// TIA Portal V17 export
// export: Created 2025-05-08T13:17:39.9382166Z, ExportSetting WithDefaults, DisplayName Totally Integrated Automation Portal, DisplayVersion V17 Update 8, DisplayName TIA Portal Openness, DisplayVersion V17 Update 8, DisplayName TIA Portal Version Control Interface, DisplayVersion V17, DisplayName SINAMICS Startdrive Advanced, DisplayVersion V17 SP2, DisplayName SINAMICS Startdrive G110M, G120, G120C, G120D, G120P, G115D, DisplayVersion V17 SP2, DisplayName SINAMICS Startdrive G130, G150, S120, S150, SINAMICS MV, S210, DisplayVersion V17 SP2, DisplayName STEP 7 Professional, DisplayVersion V17 Update 8, DisplayName SINUMERIK ONE STEP 7 Toolbox, DisplayVersion V17 Update 12, DisplayName SINUMERIK 840D sl STEP 7 Toolbox, DisplayVersion V17 Update 12, DisplayName STEP 7 Safety, DisplayVersion V17 Update 6, DisplayName WinCC Advanced, DisplayVersion V17 Update 8
FUNCTION "FC2011_STEP_BY_STEP_MODE" : Void   // FC2011, LAD
{ S7_Optimized_Access := 'FALSE' }
AUTHOR : ETXETAR
VERSION : 1.0
// stored: AutoNumber false, IsIECCheckEnabled false, SetENOAutomatically false, UDAEnableTagReadback false
   VAR CONSTANT
      FC_NUMBER : DInt := 2011;
   END_VAR
   VAR_TEMP   // added for the SCL form of the ladder/FBD networks
      _w1 : Bool;
      _w2 : Bool;
   END_VAR
BEGIN

REGION Network 1: GENERAL CONDITIONS
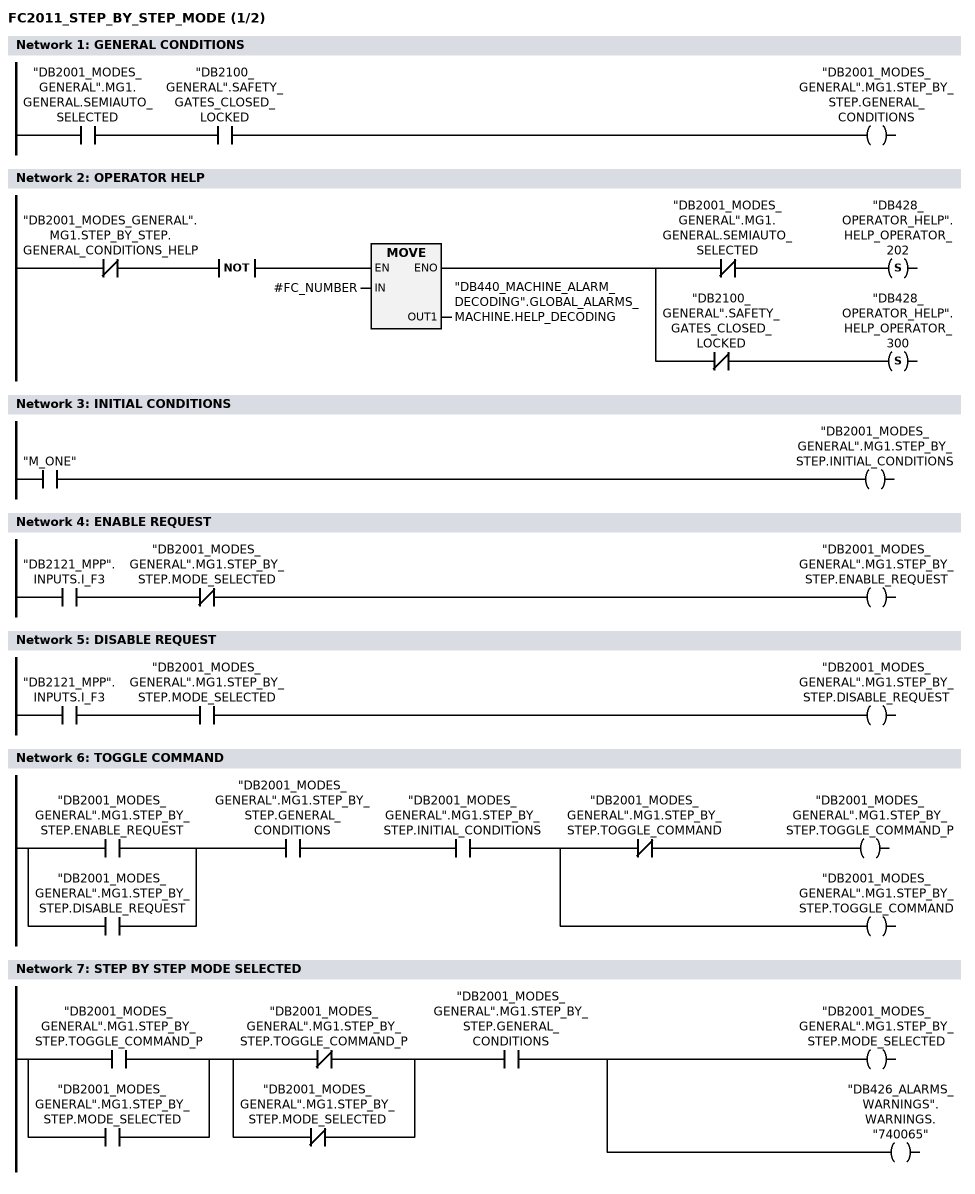
   RUNG wire#powerrail
      Contact( "DB2001_MODES_GENERAL".MG1.GENERAL.SEMIAUTO_SELECTED )
      Contact( "DB2100_GENERAL".SAFETY_GATES_CLOSED_LOCKED )
      Coil( "DB2001_MODES_GENERAL".MG1.STEP_BY_STEP.GENERAL_CONDITIONS )
   END_RUNG
   // the same network as SCL:
   "DB2001_MODES_GENERAL".MG1.STEP_BY_STEP.GENERAL_CONDITIONS := "DB2001_MODES_GENERAL".MG1.GENERAL.SEMIAUTO_SELECTED AND "DB2100_GENERAL".SAFETY_GATES_CLOSED_LOCKED;
END_REGION

REGION Network 2: OPERATOR HELP
   RUNG wire#powerrail
      I_Contact( "DB2001_MODES_GENERAL".MG1.STEP_BY_STEP.GENERAL_CONDITIONS_HELP )
      Not()
      { S7_GenerateENO := "TRUE" } Move(in := #FC_NUMBER, out1 => "DB440_MACHINE_ALARM_DECODING".GLOBAL_ALARMS_MACHINE.HELP_DECODING)
      wire#w1
      I_Contact( "DB2001_MODES_GENERAL".MG1.GENERAL.SEMIAUTO_SELECTED )
      S_Coil( "DB428_OPERATOR_HELP".HELP_OPERATOR_202 )
   END_RUNG
   RUNG wire#w1
      I_Contact( "DB2100_GENERAL".SAFETY_GATES_CLOSED_LOCKED )
      S_Coil( "DB428_OPERATOR_HELP".HELP_OPERATOR_300 )
   END_RUNG
   // the same network as SCL:
   // ENO of a box is taken as its EN; it also drops when the box reports an error
   #_w1 := NOT (NOT "DB2001_MODES_GENERAL".MG1.STEP_BY_STEP.GENERAL_CONDITIONS_HELP);
   IF #_w1 THEN "DB440_MACHINE_ALARM_DECODING".GLOBAL_ALARMS_MACHINE.HELP_DECODING := #FC_NUMBER; END_IF;
   IF #_w1 AND NOT "DB2001_MODES_GENERAL".MG1.GENERAL.SEMIAUTO_SELECTED THEN
       "DB428_OPERATOR_HELP".HELP_OPERATOR_202 := TRUE;
   END_IF;
   IF #_w1 AND NOT "DB2100_GENERAL".SAFETY_GATES_CLOSED_LOCKED THEN
       "DB428_OPERATOR_HELP".HELP_OPERATOR_300 := TRUE;
   END_IF;
END_REGION

REGION Network 3: INITIAL CONDITIONS
   RUNG wire#powerrail
      Contact( "M_ONE" )
      Coil( "DB2001_MODES_GENERAL".MG1.STEP_BY_STEP.INITIAL_CONDITIONS )
   END_RUNG
   // the same network as SCL:
   "DB2001_MODES_GENERAL".MG1.STEP_BY_STEP.INITIAL_CONDITIONS := "M_ONE";
END_REGION

REGION Network 4: ENABLE REQUEST
   RUNG wire#powerrail
      Contact( "DB2121_MPP".INPUTS.I_F3 )
      I_Contact( "DB2001_MODES_GENERAL".MG1.STEP_BY_STEP.MODE_SELECTED )
      Coil( "DB2001_MODES_GENERAL".MG1.STEP_BY_STEP.ENABLE_REQUEST )
   END_RUNG
   // the same network as SCL:
   "DB2001_MODES_GENERAL".MG1.STEP_BY_STEP.ENABLE_REQUEST := "DB2121_MPP".INPUTS.I_F3 AND NOT "DB2001_MODES_GENERAL".MG1.STEP_BY_STEP.MODE_SELECTED;
END_REGION

REGION Network 5: DISABLE REQUEST
   RUNG wire#powerrail
      Contact( "DB2121_MPP".INPUTS.I_F3 )
      Contact( "DB2001_MODES_GENERAL".MG1.STEP_BY_STEP.MODE_SELECTED )
      Coil( "DB2001_MODES_GENERAL".MG1.STEP_BY_STEP.DISABLE_REQUEST )
   END_RUNG
   // the same network as SCL:
   "DB2001_MODES_GENERAL".MG1.STEP_BY_STEP.DISABLE_REQUEST := "DB2121_MPP".INPUTS.I_F3 AND "DB2001_MODES_GENERAL".MG1.STEP_BY_STEP.MODE_SELECTED;
END_REGION

REGION Network 6: TOGGLE COMMAND
   RUNG wire#powerrail
      Contact( "DB2001_MODES_GENERAL".MG1.STEP_BY_STEP.ENABLE_REQUEST )
      wire#w1
      Contact( "DB2001_MODES_GENERAL".MG1.STEP_BY_STEP.GENERAL_CONDITIONS )
      Contact( "DB2001_MODES_GENERAL".MG1.STEP_BY_STEP.INITIAL_CONDITIONS )
      wire#w2
      I_Contact( "DB2001_MODES_GENERAL".MG1.STEP_BY_STEP.TOGGLE_COMMAND )
      Coil( "DB2001_MODES_GENERAL".MG1.STEP_BY_STEP.TOGGLE_COMMAND_P )
   END_RUNG
   RUNG wire#powerrail
      Contact( "DB2001_MODES_GENERAL".MG1.STEP_BY_STEP.DISABLE_REQUEST )
   END_RUNG wire#w1
   RUNG wire#w2
      Coil( "DB2001_MODES_GENERAL".MG1.STEP_BY_STEP.TOGGLE_COMMAND )
   END_RUNG
   // the same network as SCL:
   #_w1 := ("DB2001_MODES_GENERAL".MG1.STEP_BY_STEP.ENABLE_REQUEST OR "DB2001_MODES_GENERAL".MG1.STEP_BY_STEP.DISABLE_REQUEST) AND "DB2001_MODES_GENERAL".MG1.STEP_BY_STEP.GENERAL_CONDITIONS AND "DB2001_MODES_GENERAL".MG1.STEP_BY_STEP.INITIAL_CONDITIONS;
   "DB2001_MODES_GENERAL".MG1.STEP_BY_STEP.TOGGLE_COMMAND_P := #_w1 AND NOT "DB2001_MODES_GENERAL".MG1.STEP_BY_STEP.TOGGLE_COMMAND;
   "DB2001_MODES_GENERAL".MG1.STEP_BY_STEP.TOGGLE_COMMAND := #_w1;
END_REGION

REGION Network 7: STEP BY STEP MODE SELECTED
   RUNG wire#powerrail
      Contact( "DB2001_MODES_GENERAL".MG1.STEP_BY_STEP.TOGGLE_COMMAND_P )
      wire#w1
      I_Contact( "DB2001_MODES_GENERAL".MG1.STEP_BY_STEP.TOGGLE_COMMAND_P )
      wire#w2
      Contact( "DB2001_MODES_GENERAL".MG1.STEP_BY_STEP.GENERAL_CONDITIONS )
      wire#w3
      Coil( "DB2001_MODES_GENERAL".MG1.STEP_BY_STEP.MODE_SELECTED )
   END_RUNG
   RUNG wire#powerrail
      Contact( "DB2001_MODES_GENERAL".MG1.STEP_BY_STEP.MODE_SELECTED )
   END_RUNG wire#w1
   RUNG wire#w1
      I_Contact( "DB2001_MODES_GENERAL".MG1.STEP_BY_STEP.MODE_SELECTED )
   END_RUNG wire#w2
   RUNG wire#w3
      Coil( "DB426_ALARMS_WARNINGS".WARNINGS."740065" )
   END_RUNG
   // the same network as SCL:
   "DB2001_MODES_GENERAL".MG1.STEP_BY_STEP.MODE_SELECTED := ("DB2001_MODES_GENERAL".MG1.STEP_BY_STEP.TOGGLE_COMMAND_P OR "DB2001_MODES_GENERAL".MG1.STEP_BY_STEP.MODE_SELECTED) AND (NOT "DB2001_MODES_GENERAL".MG1.STEP_BY_STEP.TOGGLE_COMMAND_P OR NOT "DB2001_MODES_GENERAL".MG1.STEP_BY_STEP.MODE_SELECTED) AND "DB2001_MODES_GENERAL".MG1.STEP_BY_STEP.GENERAL_CONDITIONS;
   "DB426_ALARMS_WARNINGS".WARNINGS."740065" := "DB2001_MODES_GENERAL".MG1.STEP_BY_STEP.MODE_SELECTED;
END_REGION

REGION Network 8: WARNINGS
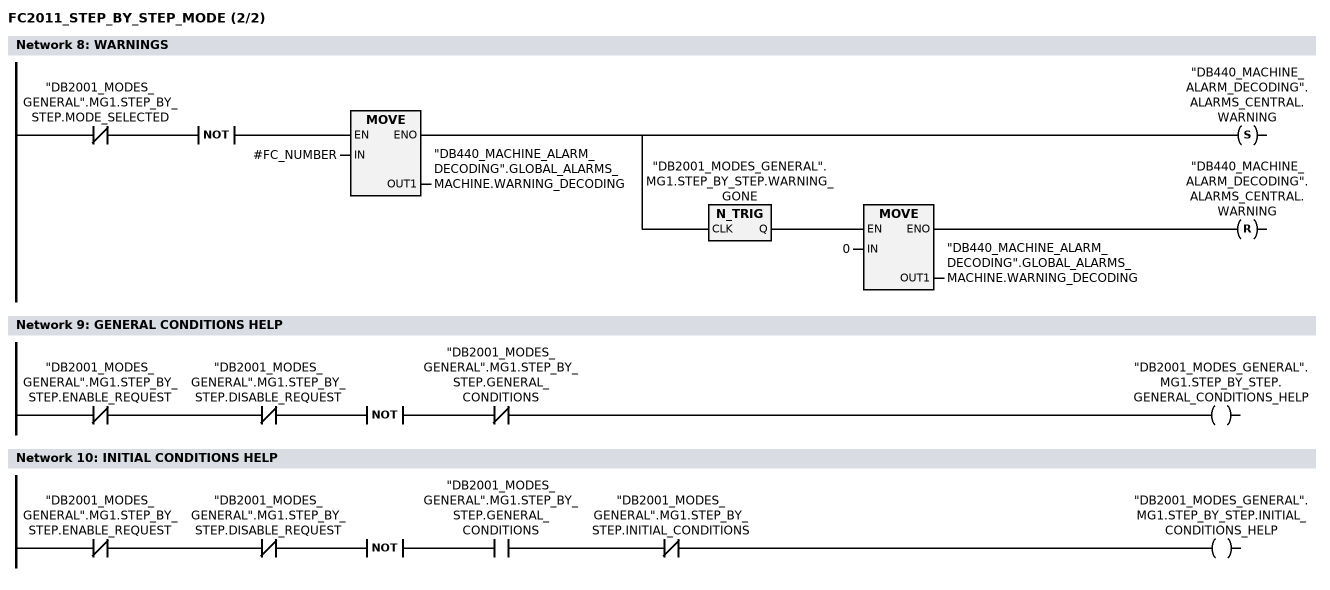
   RUNG wire#powerrail
      I_Contact( "DB2001_MODES_GENERAL".MG1.STEP_BY_STEP.MODE_SELECTED )
      Not()
      Move(in := #FC_NUMBER, out1 => "DB440_MACHINE_ALARM_DECODING".GLOBAL_ALARMS_MACHINE.WARNING_DECODING)
      wire#w1
      S_Coil( "DB440_MACHINE_ALARM_DECODING".ALARMS_CENTRAL.WARNING )
   END_RUNG
   RUNG wire#w1
      N_Trig( "DB2001_MODES_GENERAL".MG1.STEP_BY_STEP.WARNING_GONE )
      Move(in := 0, out1 => "DB440_MACHINE_ALARM_DECODING".GLOBAL_ALARMS_MACHINE.WARNING_DECODING)
      R_Coil( "DB440_MACHINE_ALARM_DECODING".ALARMS_CENTRAL.WARNING )
   END_RUNG
   // the same network as SCL:
   #_w1 := NOT (NOT "DB2001_MODES_GENERAL".MG1.STEP_BY_STEP.MODE_SELECTED);
   IF #_w1 THEN
       "DB440_MACHINE_ALARM_DECODING".GLOBAL_ALARMS_MACHINE.WARNING_DECODING := #FC_NUMBER;
       "DB440_MACHINE_ALARM_DECODING".ALARMS_CENTRAL.WARNING := TRUE;
   END_IF;
   #_w2 := NOT #_w1 AND "DB2001_MODES_GENERAL".MG1.STEP_BY_STEP.WARNING_GONE;   // falling edge
   "DB2001_MODES_GENERAL".MG1.STEP_BY_STEP.WARNING_GONE := #_w1;
   IF #_w2 THEN
       "DB440_MACHINE_ALARM_DECODING".GLOBAL_ALARMS_MACHINE.WARNING_DECODING := 0;
       "DB440_MACHINE_ALARM_DECODING".ALARMS_CENTRAL.WARNING := FALSE;
   END_IF;
END_REGION

REGION Network 9: GENERAL CONDITIONS HELP
   RUNG wire#powerrail
      I_Contact( "DB2001_MODES_GENERAL".MG1.STEP_BY_STEP.ENABLE_REQUEST )
      I_Contact( "DB2001_MODES_GENERAL".MG1.STEP_BY_STEP.DISABLE_REQUEST )
      Not()
      I_Contact( "DB2001_MODES_GENERAL".MG1.STEP_BY_STEP.GENERAL_CONDITIONS )
      Coil( "DB2001_MODES_GENERAL".MG1.STEP_BY_STEP.GENERAL_CONDITIONS_HELP )
   END_RUNG
   // the same network as SCL:
   "DB2001_MODES_GENERAL".MG1.STEP_BY_STEP.GENERAL_CONDITIONS_HELP := NOT (NOT "DB2001_MODES_GENERAL".MG1.STEP_BY_STEP.ENABLE_REQUEST AND NOT "DB2001_MODES_GENERAL".MG1.STEP_BY_STEP.DISABLE_REQUEST) AND NOT "DB2001_MODES_GENERAL".MG1.STEP_BY_STEP.GENERAL_CONDITIONS;
END_REGION

REGION Network 10: INITIAL CONDITIONS HELP
   RUNG wire#powerrail
      I_Contact( "DB2001_MODES_GENERAL".MG1.STEP_BY_STEP.ENABLE_REQUEST )
      I_Contact( "DB2001_MODES_GENERAL".MG1.STEP_BY_STEP.DISABLE_REQUEST )
      Not()
      Contact( "DB2001_MODES_GENERAL".MG1.STEP_BY_STEP.GENERAL_CONDITIONS )
      I_Contact( "DB2001_MODES_GENERAL".MG1.STEP_BY_STEP.INITIAL_CONDITIONS )
      Coil( "DB2001_MODES_GENERAL".MG1.STEP_BY_STEP.INITIAL_CONDITIONS_HELP )
   END_RUNG
   // the same network as SCL:
   "DB2001_MODES_GENERAL".MG1.STEP_BY_STEP.INITIAL_CONDITIONS_HELP := NOT (NOT "DB2001_MODES_GENERAL".MG1.STEP_BY_STEP.ENABLE_REQUEST AND NOT "DB2001_MODES_GENERAL".MG1.STEP_BY_STEP.DISABLE_REQUEST) AND "DB2001_MODES_GENERAL".MG1.STEP_BY_STEP.GENERAL_CONDITIONS AND NOT "DB2001_MODES_GENERAL".MG1.STEP_BY_STEP.INITIAL_CONDITIONS;
END_REGION
END_FUNCTION
